PROGRAM MAIN
VAR
END_VAR

END_PROGRAM

(* stored: Version 1.1.0.1
   POU MAIN: Id {ee19d2c5-6dc6-40b9-bf87-3b738561f38e} *)
